// TwinCAT 3 PLC project DCSv1
// ProgramVersion: 3.1.4023.0
// libraries:
//   Tc2_MC2, * (Beckhoff Automation GmbH)
//   Tc2_MC2_Drive, * (Beckhoff Automation GmbH)
//   Tc2_SerialCom, * (Beckhoff Automation GmbH)
//   Tc2_Standard, * (Beckhoff Automation GmbH)
//   Tc2_System, * (Beckhoff Automation GmbH)
//   Tc3_Module, * (Beckhoff Automation GmbH)
// project tree:
//   / ComTask.TcTTO (not stored), PlcTask.TcTTO (not stored)
//   GVLs/GVLs/ GVL.TcGVL, GVL_IO.TcGVL, GVL_ResearchData.TcGVL, GVL_VAR.TcGVL, ReadMe.TcGVL
//   POUs/FB/ FB_Analog.TcPOU (not stored), F_ScalAnalogOut.TcPOU
//   POUs/ MAIN.TcPOU, P_AP1_Check.TcPOU, P_ComEL6001.TcPOU (not stored), P_CP1_Calibration.TcPOU, P_CP1_Enable.TcPOU (not stored), P_MI1_OnOff.TcPOU (not stored), P_AP1_OnOff.TcPOU (not stored), P_ModeSelector.TcPOU, P_Outputs_Manual.TcPOU, P_Set_Research_Data.TcPOU, P_Read_Research_Data.TcPOU, P_SP1_Check.TcPOU, P_SP1_OnOff.TcPOU
//   POUs/POUs/ FB_Drive.TcPOU (not stored), FB_Mixer1_2.TcPOU
// real-time tasks:
//   TASK PlcTask: cycle T#10ms, priority 20, ADS port 350
//   TASK ComTask: cycle T#10ms, priority 21, ADS port 351
// motion (NC):
//   TASK NC-Task 1 SAF: cycle T#2ms, priority 4, ADS port 501
//   TASK NC-Task 1 SVB: cycle T#10ms, priority 8, ADS port 511
//   AXIS Mixer 1 (id 2)
//     General: UnitName=°, UnitFlags=#x00000004
//     Dynamic: Acceleration=7443.34, Deceleration=7443.34, Jerk=22330
//     Velo: RefSearch=49.6222741699219, RefSync=49.6222741699219, SlowManual=248.111370849609, FastManual=1488.66822509766, Fast=4962.22741699219, Maximum=4962.23
//     OtherSettings: AllowMotionCmdToSlave=true
//     encoder EncType=8
//       EncPara: ScaleFactorNumerator=45, ScaleFactorDenominator=1048576, Offset=-131121.7408, Inverse=true, MaxCount=#x007fffff, ReferenceSystem=2
//     drive DrvType=9
//       DrvPara: Inverse=true, MaxCount=#xffffffff, DriveControlDWord=#x00030100
//         Analog: VeloReferenz=5458.45015869141, VeloScale=1.02400649589962, ScaleFactorActTorque=0.1
//         TimeComp: TaskDelayCycles=1
//     controller CtrType=1
//       CtrPara: PriorControlFactor=1
//         Observer: BandWidth=20
//   AXIS Mixer 2 (id 3)
//     General: UnitName=°, UnitFlags=#x00000004
//     Dynamic: Acceleration=7443.34112548828, Deceleration=7443.34112548828, Jerk=22330.0233764648
//     Velo: RefSearch=49.6222741699219, RefSync=49.6222741699219, SlowManual=248.111370849609, FastManual=1488.66822509766, Fast=4962.22741699219, Maximum=4962.22741699219
//     OtherSettings: AllowMotionCmdToSlave=true
//     encoder EncType=8
//       EncPara: ScaleFactorNumerator=45, ScaleFactorDenominator=1048576, MaxCount=#x007fffff, ReferenceSystem=2
//     drive DrvType=9
//       DrvPara: MaxCount=#xffffffff, DriveControlDWord=#x00030100
//         Analog: VeloReferenz=5458.45015869141, VeloScale=1.02400649589962, ScaleFactorActTorque=0.1
//         TimeComp: TaskDelayCycles=1
//     controller CtrType=1
//       CtrPara: PriorControlFactor=1
//         Observer: BandWidth=20
// I/O:
//   DEVICE Device 1 (EtherCAT), AmsNetId 172.17.147.1.3.1
//     Term 1 (EK1200) [EK1200-5000 EtherCAT Power supply (2A E-Bus)]
//       Term 2 (EL1008) 30K3 [EL1008 8Ch. Dig. Input 24V, 3ms]
//       Term 3 (EL1008) 30K3.1 [EL1008 8Ch. Dig. Input 24V, 3ms]
//       Term 10 (EL1008) new [EL1008 8Ch. Dig. Input 24V, 3ms]
//       Term 4 (EL2008) 30K4 [EL2008 8Ch. Dig. Output 24V, 0.5A]
//       Term 5 (EL2008) 30K5 [EL2008 8Ch. Dig. Output 24V, 0.5A]
//       Term 12 (EL2008) new [EL2008 8Ch. Dig. Output 24V, 0.5A]
//       Term 13 (EL3022) new [EL3022 2Ch. Ana. Input 4-20mA DIFF]
//       Term 14 (EL3202) new [EL3202 2Ch. Ana. Input PT100 (RTD)]
//       Term 6 (EL3255) 30K5.1 [EL3255 5Ch. potentiometer measurement with sensor supply]
//       Term 7 (EL4134) 30K6 [EL4134 4Ch. Ana. Output -10/+10V, 16bit]
//       Term 8 (EL6001) [EL6001 Interface (RS232)]
//       Term 15 (EL6631) new [EL6631 PROFINET IO Controller]
//       Term 9 (EL9011) [EL9011 End Terminal]
//   DEVICE Device 4 (EtherCAT), AmsNetId 172.17.147.1.5.1
//     Drive 11 (AX5206-0000-0213) [AX5206-0000-0213 EtherCAT Drive (SoE, 2 Ch.)]
// variable links:
//   NC-Task 1 SAF/Axes/Mixer 1 <-> Device 4 (EtherCAT)/Drive 11 (AX5206-0000-0213)
//     Drive/Inputs/In/nDataIn1 <-> AT 1/Following distance
//     Drive/Inputs/In/nDcOutputTime <-> InfoData/DcOutputShift
//     Drive/Inputs/In/nState1 <-> AT 1/Drive status word @bit 8
//     Drive/Inputs/In/nState2 <-> AT 1/Drive status word
//     Drive/Inputs/In/nState4 @bit 1 <-> WcState/InputToggle
//     Drive/Inputs/In/nState4 <-> WcState/WcState
//     Drive/Outputs/Out/nCtrl1 <-> MDT 1/Master control word @bit 8
//     Drive/Outputs/Out/nDataOut1 <-> MDT 1/Position command value
//     Enc/Inputs/In/nDataIn1 <-> AT 1/Position feedback 1 value
//     Enc/Inputs/In/nDcInputTime <-> InfoData/DcInputShift
//     Enc/Inputs/In/nState4 @bit 1 <-> WcState/InputToggle
//     Enc/Inputs/In/nState4 <-> WcState/WcState
//   NC-Task 1 SAF/Axes/Mixer 2 <-> Device 4 (EtherCAT)/Drive 11 (AX5206-0000-0213)
//     Drive/Inputs/In/nDataIn1 <-> AT 2/Following distance
//     Drive/Inputs/In/nDcOutputTime <-> InfoData/DcOutputShift
//     Drive/Inputs/In/nState1 <-> AT 2/Drive status word @bit 8
//     Drive/Inputs/In/nState2 <-> AT 2/Drive status word
//     Drive/Inputs/In/nState4 @bit 1 <-> WcState/InputToggle
//     Drive/Inputs/In/nState4 <-> WcState/WcState
//     Drive/Outputs/Out/nCtrl1 <-> MDT 2/Master control word @bit 8
//     Drive/Outputs/Out/nDataOut1 <-> MDT 2/Position command value
//     Enc/Inputs/In/nDataIn1 <-> AT 2/Position feedback 1 value
//     Enc/Inputs/In/nDcInputTime <-> InfoData/DcInputShift
//     Enc/Inputs/In/nState4 @bit 1 <-> WcState/InputToggle
//     Enc/Inputs/In/nState4 <-> WcState/WcState
//   DCSv1/DCSv1 Instance <-> Device 1 (EtherCAT)/Term 1 (EK1200)/Term 10 (EL1008) new
//     PlcTask Inputs/GVL_IO.ib_SP1_No_Error <-> Channel 2/Input
//     PlcTask Inputs/GVL_IO.ib_SP1_Ready <-> Channel 1/Input
//   DCSv1/DCSv1 Instance <-> Device 1 (EtherCAT)/Term 1 (EK1200)/Term 2 (EL1008) 30K3
//     ComTask Inputs/GVL_IO.ib_CP1_Ready <-> Channel 3/Input
//     PlcTask Inputs/GVL_IO.ib_AP1_No_Error <-> Channel 6/Input
//     PlcTask Inputs/GVL_IO.ib_AP1_Ready <-> Channel 5/Input
//     PlcTask Inputs/GVL_IO.ib_CC1_Button_Mode_Laptop <-> Channel 8/Input
//     PlcTask Inputs/GVL_IO.ib_CC1_Button_Reset <-> Channel 7/Input
//     PlcTask Inputs/GVL_IO.ib_CC1_Safety_Ready <-> Channel 1/Input
//     PlcTask Inputs/GVL_IO.ib_CP1_Drive_Error <-> Channel 4/Input
//     PlcTask Inputs/GVL_IO.ib_CP1_Safety_Grid_Mounted <-> Channel 2/Input
//   DCSv1/DCSv1 Instance <-> Device 1 (EtherCAT)/Term 1 (EK1200)/Term 3 (EL1008) 30K3.1
//     PlcTask Inputs/GVL_IO.ib_AP1_Button_Not_Off <-> Channel 7/Input
//     PlcTask Inputs/GVL_IO.ib_AP1_Button_On <-> Channel 6/Input
//     PlcTask Inputs/GVL_IO.ib_CC1_Button_Mode_Manual <-> Channel 1/Input
//     PlcTask Inputs/GVL_IO.ib_MI1_Button_Not_Off <-> Channel 3/Input
//     PlcTask Inputs/GVL_IO.ib_MI1_Button_On <-> Channel 2/Input
//     PlcTask Inputs/GVL_IO.ib_SP1_Button_Not_Off <-> Channel 5/Input
//     PlcTask Inputs/GVL_IO.ib_SP1_Button_On <-> Channel 4/Input
//   DCSv1/DCSv1 Instance <-> Device 1 (EtherCAT)/Term 1 (EK1200)/Term 4 (EL2008) 30K4
//     PlcTask Outputs/GVL_IO.ob_AP1_Pressure_Ok <-> Channel 7/Output
//     PlcTask Outputs/GVL_IO.ob_AP1_Pulse <-> Channel 8/Output
//     PlcTask Outputs/GVL_IO.ob_AP1_Start <-> Channel 6/Output
//     PlcTask Outputs/GVL_IO.ob_CC1_Safety_Reset <-> Channel 1/Output
//     PlcTask Outputs/GVL_IO.ob_CP1_Backward <-> Channel 5/Output
//     PlcTask Outputs/GVL_IO.ob_CP1_Forward <-> Channel 4/Output
//     PlcTask Outputs/GVL_IO.ob_CP1_Start <-> Channel 3/Output
//     PlcTask Outputs/GVL_IO.ob_CP1_Stop <-> Channel 2/Output
//   DCSv1/DCSv1 Instance <-> Device 1 (EtherCAT)/Term 1 (EK1200)/Term 5 (EL2008) 30K5
//     PlcTask Outputs/GVL_IO.ob_AP1_Not_Empty <-> Channel 1/Output
//     PlcTask Outputs/GVL_IO.ob_AP1_Power_On <-> Channel 2/Output
//     PlcTask Outputs/GVL_IO.ob_SP1_Not_Empty <-> Channel 6/Output
//     PlcTask Outputs/GVL_IO.ob_SP1_Power_On <-> Channel 7/Output
//     PlcTask Outputs/GVL_IO.ob_SP1_Pressure_Ok <-> Channel 4/Output
//     PlcTask Outputs/GVL_IO.ob_SP1_Pulse <-> Channel 5/Output
//     PlcTask Outputs/GVL_IO.ob_SP1_Start <-> Channel 3/Output
//   DCSv1/DCSv1 Instance <-> Device 1 (EtherCAT)/Term 1 (EK1200)/Term 6 (EL3255) 30K5.1
//     ComTask Inputs/GVL_IO.in_AP1_Poti_Speed <-> AI Standard Channel 3/Value
//     ComTask Inputs/GVL_IO.in_PP1_Poti_Speed <-> AI Standard Channel 2/Value
//     PlcTask Inputs/GVL.nInputSpare1 <-> AI Standard Channel 4/Value
//     PlcTask Inputs/GVL.nInputSpare2 <-> AI Standard Channel 5/Value
//     PlcTask Inputs/GVL_IO.in_MI1_Poti_Speed <-> AI Standard Channel 1/Value
//   DCSv1/DCSv1 Instance <-> Device 1 (EtherCAT)/Term 1 (EK1200)/Term 7 (EL4134) 30K6
//     PlcTask Outputs/GVL_IO.on_AP1_Speed <-> AO Output Channel 2/Analog output
//     PlcTask Outputs/GVL_IO.on_CP1_Speed <-> AO Output Channel 1/Analog output
//     PlcTask Outputs/GVL_IO.on_SP1_Speed <-> AO Output Channel 3/Analog output
//   DCSv1/DCSv1 Instance <-> Device 1 (EtherCAT)/Term 1 (EK1200)/Term 8 (EL6001)
//     ComTask Inputs/GVL.stIn_EL6001/D <-> COM Inputs/Data In 0
//     ComTask Inputs/GVL.stIn_EL6001/D @bit {8..168 step 8} <-> COM Inputs/Data In {1..21}  (21 links)
//     ComTask Inputs/GVL.stIn_EL6001/Status <-> COM Inputs/Status
//     ComTask Outputs/GVL.stOut_EL6001/Ctrl <-> COM Outputs/Ctrl
//     ComTask Outputs/GVL.stOut_EL6001/D <-> COM Outputs/Data Out 0
//     ComTask Outputs/GVL.stOut_EL6001/D @bit {8..168 step 8} <-> COM Outputs/Data Out {1..21}  (21 links)
//   DCSv1/DCSv1 Instance <-> Device 4 (EtherCAT)/Drive 11 (AX5206-0000-0213)
//     PlcTask Inputs/GVL.in_MID1_ActAbsCurrent <-> AT 1/Actual absolute current
//     PlcTask Inputs/GVL.in_MID2_ActAbsCurrent <-> AT 2/Actual absolute current
//     PlcTask Inputs/GVL.in_MID1_ActMotorTemperature <-> AT 1/Motor temperature
//     PlcTask Inputs/GVL.in_MID2_ActMotorTemperature <-> AT 2/Motor temperature
//   DCSv1/DCSv1 Instance <-> NC-Task 1 SAF/Axes/Mixer 1
//     PlcTask Inputs/GVL.Axis_Mixer1.NcToPlc <-> Outputs/ToPlc
//     PlcTask Outputs/GVL.Axis_Mixer1.PlcToNc <-> Inputs/FromPlc
//   DCSv1/DCSv1 Instance <-> NC-Task 1 SAF/Axes/Mixer 2
//     PlcTask Inputs/GVL.Axis_Mixer2.NcToPlc <-> Outputs/ToPlc
//     PlcTask Outputs/GVL.Axis_Mixer2.PlcToNc <-> Inputs/FromPlc

// ---- GVLs/GVLs/GVL.TcGVL
{attribute 'qualified_only'}
VAR_GLOBAL
	
	
	//
	// Data Communication RS-232
	TxBufferEL								: ComBuffer;
	RxBufferEL								: ComBuffer;
	
			
	//
	// Data Communication Axis Mixers

	//
	// Mixer drive A // 16.09.2021 PF
	Axis_Mixer1 							: AXIS_REF;
	f_MID1_ActCurrent: REAL;
	f_MID1_ActTorque: REAL;
	in_MID1_ActAbsCurrent AT %I*: INT;
	in_MID1_ActMotorTemperature AT %I* :INT; // 220817 WT 
	
	//
	// Mixer drive B // 16.09.2021 PF
	Axis_Mixer2 							: AXIS_REF;
	f_MID2_ActCurrent: REAL;
	f_MID2_ActTorque: REAL;
	in_MID2_ActAbsCurrent AT %I*: INT;
	in_MID2_ActMotorTemperature AT %I* :INT; // 220817 WT
	
	//
	// Control Input Speed
	fControlMixerPumpSpeed					: REAL; 
	fControlPeristalticPumpSpeed			: REAL; 
	fControlDosingPumpSpeed					: REAL; 
	fInputSpare1							: REAL; 
	fInputSpare2							: REAL; 
	
	//
	// Output Speed
	fConcretePumpSpeed						: REAL;
	fDosingPumpSpeed						: REAL;
	fOutputSpare1							: REAL;
	fOutputSpare2							: REAL;
	
	
	//
	//Hardware Input
	bSafetyIO						AT %I*	: BOOL;
	// bConcretePumpSafetyGridMounted	AT %I*	: BOOL;
	// bConcretePumpReady				AT %I*	: BOOL;
	// bConcretePumpFcError				AT %I*	: BOOL;
	bDosingPumpReady				AT %I*	: BOOL;
	bDosingPumpNoError				AT %I*	: BOOL;
	bControlResetSafety				AT %I*	: BOOL;
	bControlLaptop					AT %I*	: BOOL;
	bControlManual					AT %I*	: BOOL;	
	nControlMixerPumpOn				AT %I*	: BOOL; 
	nControlMixerPumpOff			AT %I*	: BOOL; 
	nControlConcretPumpOn			AT %I*	: BOOL; 
	nControlConcretPumpOff			AT %I*	: BOOL; 
	nControlDosingPumpOn			AT %I*	: BOOL; 
	nControlDosingPumpOff			AT %I*	: BOOL; 
	bInputSpare1					AT %I*	: BOOL;
		
	nControlMixerPumpSpeed			AT %I*	: INT; 
	// nControlPeristalticPumpSpeed	AT %I*	: INT; 
	nControlDosingPumpSpeed			AT %I*	: INT; 
	nInputSpare1					AT %I*	: INT; 
	nInputSpare2					AT %I*	: INT; 

	
	//
	//Hardware Output
	bResetSafety					AT %Q*	: BOOL;
	// bConcretePumpOn					AT %Q*	: BOOL;
	// bConcretePumpOff					AT %Q*	: BOOL;
	// bConcretePumpForwardOn			AT %Q*	: BOOL;
	// bConcretePumpBackwardOn			AT %Q*	: BOOL;
	bDosingPumpDosingHighLow		AT %Q*	: BOOL;
	bDosingPumpNoFastStop			AT %Q*	: BOOL;
	bDosingPumpDosingAmount			AT %Q*	: BOOL;
	bOutputSpare1					AT %Q*	: BOOL;
	bOutputSpare2					AT %Q*	: BOOL;
	bOutputSpare3					AT %Q*	: BOOL;
	bOutputSpare4					AT %Q*	: BOOL;
	bOutputSpare5					AT %Q*	: BOOL;
	bOutputSpare6					AT %Q*	: BOOL;
	bOutputSpare7					AT %Q*	: BOOL;
	bOutputSpare8					AT %Q*	: BOOL;
	
	// nConcretePumpSpeed				AT %Q*	: INT;
	nDosingPumpSpeed				AT %Q*	: INT;
	nOutputSpare1					AT %Q*	: INT;
	nOutputSpare2					AT %Q*	: INT;
	
	
	//
	//Hardware RS-232
	stIn_EL6001 					AT %I*	: EL6inData22B;	
	stOut_EL6001 					AT %Q*	: EL6outData22B;
	
END_VAR

// ---- GVLs/GVLs/GVL_IO.TcGVL
{attribute 'qualified_only'}
VAR_GLOBAL
//***********************************************************************************
//
// ETH Zürich / Robotic Fabrication Lab
// HIB C 13 / Stefano-Franscini-Platz 1
// CH-8093 Zürich
// 
// ***********************************************************************************
// 
// PROJECT     :  A061 Inline Mixer
// 
// FUNCTION    :  Global Varable In and Outputs
// 
// AUTHOR      :  Fabio Scotto / Philippe Fleischmann
// 
// EMAIL       :  scotto@arch.ethz.ch / fleischmann@arch.ehtz.ch
// 
// Copyright   :  ETH Zürich (CH) 2020
//
// ***********************************************************************************

//
// Inputs

//
// Concrete Controller 1
ib_CC1_Safety_Ready AT %I*: BOOL;
ib_CC1_Button_Mode_Manual AT %I*: BOOL;
ib_CC1_Button_Mode_Laptop AT %I*: BOOL;
//ib_CC1_Button_Mode_Robot AT %I*:BOOL;
//
ib_CC1_Button_Reset AT %I*: BOOL;

//
// Concrete Pump 1
ib_CP1_Drive_Error AT %I*: BOOL;
ib_CP1_Ready AT %I*: BOOL;
ib_CP1_Safety_Grid_Mounted AT %I*: BOOL;
in_CP1_Tube_Pressure_Sensor AT %I*: INT;
in_CP1_Tube_Temperature_Sensor AT %I*: INT;

//
// Peristaltic Pump 1 ( SHOULD BE REMOVE, it is old pump 
in_PP1_Poti_Speed AT %I*	: INT; 

//
// Accelerator Pump 1
ib_AP1_Button_On AT %I*: BOOL;
ib_AP1_Button_Not_Off AT %I*: BOOL;
ib_AP1_Ready AT %I*: BOOL;
ib_AP1_No_Error AT %I*: BOOL;
in_AP1_Poti_Speed AT %I*	: INT; 

// 
// Superplasticizer Pump 1 (WT 220915)
ib_SP1_Button_On AT %I*: BOOL;
ib_SP1_Button_Not_Off AT %I*: BOOL;
ib_SP1_Ready AT %I*: BOOL;
ib_SP1_No_Error AT %I*: BOOL;
ib_SP1_Poti_Speed AT %I*: INT; 

//
// Mixer 1
ib_MI1_Button_On AT %I*: BOOL;
ib_MI1_Button_Not_Off AT %I*: BOOL;
in_MI1_Poti_Speed AT %I*	: INT; 

//
// Outputs

//
// Concrete Controller 1
ob_CC1_Safety_Reset AT %Q*: BOOL;

//
// Concrete Pump 1
ob_CP1_Start AT %Q*: BOOL;
ob_CP1_Stop AT %Q*: BOOL;
ob_CP1_Forward AT %Q*: BOOL;
ob_CP1_Backward AT %Q*: BOOL;

on_CP1_Speed AT %Q*: INT;

//
// Accelerator Pump 1
ob_AP1_Power_On AT %Q*: BOOL;
ob_AP1_Start AT %Q*: BOOL;
ob_AP1_Pressure_Ok AT %Q*: BOOL;
ob_AP1_Not_Empty AT %Q*: BOOL;
ob_AP1_Pulse AT %Q*: BOOL;

on_AP1_Speed AT %Q*: INT;

// 
// Superplasticizer Pump 1 (WT 220915)
ob_SP1_Power_On AT %Q*: BOOL;
ob_SP1_Start AT %Q*: BOOL;
ob_SP1_Pressure_Ok AT %Q*: BOOL;
ob_SP1_Not_Empty AT %Q*: BOOL;
ob_SP1_Pulse AT %Q*: BOOL;

on_SP1_Speed AT %Q*: INT;


END_VAR

// ---- GVLs/GVLs/GVL_ResearchData.TcGVL
{attribute 'qualified_only'}
VAR_GLOBAL
//***********************************************************************************
//
// ETH Zürich / Robotic Fabrication Lab
// HIB C 13 / Stefano-Franscini-Platz 1
// CH-8093 Zürich
// 
// ***********************************************************************************
// 
// PROJECT     :  A061 Inline Mixer
// 
// FUNCTION    :  Global Varable to collect all research data
// 
// AUTHOR      :  Seyma Gürel / Philippe Fleischmann / Weiting Chen
// 
// EMAIL       :  scotto@arch.ethz.ch / fleischmann@arch.ehtz.ch
// 
// Copyright   :  ETH Zürich (CH) 2021
//
// ***********************************************************************************


// ***********************************************************************************
// Process inputs
// ***********************************************************************************

//
// Mode
b_RED_Mode_Manual: BOOL; //0916 WT
b_RED_Mode_Laptop: BOOL; //0916 WT

//
// Maximal speed for mixer [°/s]  (WT 220916
f_RED_Control_Speed : LREAL;					// [°/s]
b_RED_Laptop_speed_Conctrol: BOOL;
f_RED_Control_Speed_by_Laptop:LREAL;

//
Superplasticizer_Pump: STRING := 'Superplasticizer_Pump'; 
// 
// Superplasticizer Pump (WT 220916 
b_RED_Superplasticizer_Pump_Check_On: BOOL;
n_RED_Superplasticizer_Pump_Check_Flowrate: REAL;
n_RED_Superplasticizer_Pump_Check_Duration: TIME;

b_RED_Superplasticizer_Pump_Flush_On: BOOL;
n_RED_Superplasticizer_Pump_Flush_Speed: REAL;

f_RED_Superplasticizer_Pump_Mass: REAL;             // [g/min]
f_RED_Superplasticizer_Pump_Density: REAL;          // [g/ml]
n_RED_Superplasticizer_Pump_Flowrate: REAL;         // [ml/min]

//
ACCELERATION_PUMP: STRING := 'Acceleration_Pump';
//
// Accelerator Pump
b_RED_Acceleration_Pump_Check_On: BOOL;
n_RED_Acceleration_Pump_Check_Flowrate: REAL;
n_RED_Acceleration_Pump_Check_Duration: TIME;

b_RED_Acceleration_Pump_Flush_On: BOOL;
n_RED_Acceleration_Pump_Flush_Speed: REAL;

f_RED_Acceleration_Pump_Mass: REAL;             // [g/min]
f_RED_Acceleration_Pump_Density: REAL;          // [g/ml]
n_RED_Acceleration_Pump_Flowrate: REAL;         // [ml/min]

//
CONCRETE_PUMP: STRING := 'CONCRETE_PUMP';
// Concrete Pump
//
b_RED_Concrete_Pump_Forward_On: BOOL;
b_RED_Concrete_Pump_Backward_On: BOOL;
n_RED_Concrete_Pump_Speed: INT;					// [ 0..75rpm ]
// WT 220916
b_RED_Concrete_Pump_Calibration_On: BOOL;
n_RED_Concrete_Pump_Calibration_Speed: INT;		// [rpm]
n_RED_Concrete_Pump_Calibration_Time: TIME;


// ***********************************************************************************
// Process outpus
// ***********************************************************************************

//
MIXER: STRING := 'MIXER';
// Status mixer
//
b_RED_Status_On : BOOL;
f_RED_Status_Speed_Overide : LREAL;
f_RED_Status_Speed_Motor_1 : LREAL;
f_RED_Status_Speed_Motor_2 : LREAL;
f_RED_Status_Torque_Motor_1 : REAL;				// [Nm]
f_RED_Status_Torque_Motor_2 : REAL;				// [Nm]

f_RED_Status_Temperature_Motor_1 : REAL; // [°C] 
f_RED_Status_Temperature_Motor_2 : REAL; // [°C] 

//
// Superplasticizer Pump (WT 220916
n_RED_Status_Superplasticizer_Pump_Flowrate: INT;          // [ml/min]
f_RED_Status_Superplasticizer_Pump_Max_Flowrate_ml_per_min: REAL;           // [ml/min]

//
// Accelerator Pump
n_RED_Status_Acceleration_Pump_Flowrate: INT;          // [ml/min]
f_RED_Status_Acceleration_Pump_Max_Flowrate_ml_per_min: REAL;           // [ml/min]

	n_RED_Acceleration_Pump_Calibration_Speed: INT;
	b_RED_Acceleration_Pump_Preparation_On: INT;
END_VAR

// ---- GVLs/GVLs/GVL_VAR.TcGVL
{attribute 'qualified_only'}
VAR_GLOBAL
//***********************************************************************************
//
// ETH Zürich / Robotic Fabrication Lab
// HIB C 13 / Stefano-Franscini-Platz 1
// CH-8093 Zürich
// 
// ***********************************************************************************
// 
// PROJECT     :  A061 Inline Mixer
// 
// FUNCTION    :  Global Varable In and Outputs
// 
// AUTHOR      :  Fabio Scotto / Philippe Fleischmann / Weiting Chen
// 
// EMAIL       :  scotto@arch.ethz.ch / fleischmann@arch.ehtz.ch
// 
// Copyright   :  ETH Zürich (CH) 2020
//
// ***********************************************************************************

//
// Concrete Controller 1
b_Mode_Manual : BOOL;
b_Mode_Laptop : BOOL;

//
// Concrete Pump 1

//
// Superplasticizer Pump 1
b_SP1_Run : BOOL;
f_SP1_Override :LREAL;

//
// Accelerator Pump 1
b_AP1_Run : BOOL;
f_AP1_Override : LREAL; 

//
// Mixer 1
b_MI1_ReadToDrive : BOOL;
b_MI1_Run : BOOL;
f_MI1_Override : LREAL; 
f_MI1_MaxSpeed : LREAL;
f_MI1_ActSpeedM1 : LREAL;
f_MI1_ActSpeedM2 : LREAL;

END_VAR

// ---- GVLs/GVLs/ReadMe.TcGVL
{attribute 'qualified_only'}
VAR_GLOBAL
//***********************************************************************************
//
// ETH Zürich / Robotic Fabrication Lab
// HIB C 13 / Stefano-Franscini-Platz 1
// CH-8093 Zürich
// 
// ***********************************************************************************
// 
// PROJECT     :  A061 Inline Mixer
// 
// FUNCTION    :  Read Me
// 
// AUTHOR      :  Fabio Scotto / Philippe Fleischmann
// 
// EMAIL       :  scotto@arch.ethz.ch / fleischmann@arch.ehtz.ch
// 
// Copyright   :  ETH Zürich (CH) 2020
//
// ***********************************************************************************

//
//Prefix
//ib = Input Bool   / ob = Output Bool
//if = Input float  / of = Output float (REAL, LREAL)
//in = Input numeric/ on = Outplut numerical (INT, Sint, USINT, UNIT, DINT, UDINT, BYTE, WORD, DWORD, LWORD, XINT, UXINT, XWORD) 

//
//Short Cuts
//CC1 = Concrete Controller 
//AP1 = Accelerator Pump
//CP1 = Concrete Pump
//PP1 = Peristaltic Pump
//MI1 = Mixer
//T1  = Tool 1
//CA1 = Camera 1
//RED = Research Data

END_VAR

// ---- POUs/FB/F_ScalAnalogOut.TcPOU
FUNCTION F_ScalAnalogOut : INT
VAR_INPUT
	n_Input:INT;
	n_InMin:INT;
	n_InMax:INT;
	n_OutMin:INT;
	n_OutMax:INT;

END_VAR
VAR
	f_Input:REAL;
	f_InMin:REAL;
	f_InMax:REAL;
	f_OutMin:REAL;
	f_OutMax:REAL;
	f_DeltaIn:REAL;
	f_DeltaOut:REAL;
END_VAR

//
// Convert integer to real 
f_Input:=INT_TO_REAL(n_Input);
f_InMin:=INT_TO_REAL(n_InMin);
f_InMax:=INT_TO_REAL(n_InMax);
f_OutMin:=INT_TO_REAL(n_OutMin);
f_OutMax:=INT_TO_REAL(n_OutMax);
//
// Check plausibility 
IF f_InMax = f_InMin THEN	
	//
	// Not plausible output fix value
	F_ScalAnalogOut := 0;
ELSE	
	//
	// Plausible calculate output 
	f_DeltaIn:=f_InMax-f_InMin;
	f_DeltaOut:=f_OutMax-f_OutMin;
	F_ScalAnalogOut :=REAL_TO_INT((f_DeltaOut/f_DeltaIn)*(f_Input-f_InMin));	
END_IF

END_FUNCTION

// ---- POUs/MAIN.TcPOU
PROGRAM MAIN
VAR	

	fb_MC_SetPosition		:FB_SoEAX5000SetPositionOffset;
	pos:LREAL;
	Mixer1_2		: FB_Mixer1_2;
	Analog			: FB_Analog;

	SafetyReset 	: bool;
	b_Enable		: BOOL;
	b_Reset			: BOOL;


	
	Test : MC_ReadStatus;
END_VAR

//***********************************************************************************
//
// ETH Zürich / Robotic Fabrication Lab
// HIB C 13 / Stefano-Franscini-Platz 1
// CH-8093 Zürich
// 
// ***********************************************************************************
// 
// PROJECT     :  A061 Inline Mixer
// 
// FUNCTION    :  MAIN Programm
// 
// AUTHOR      :  Mathias Suter /Weiting Chen
// 
// EMAIL       :  mathias.suter@solinaut.ch
// 
// Copyright   :  ETH Zürich (CH) 2021
//
// ***********************************************************************************


//
// Mode selector ( ONLY FOR READ OUTPUT NOW
P_ModeSelector();

//
// Set research data 
P_Set_Research_Data();

// ******************************************************************
// 220916 WT

//*************************
// Superplasticizer Pump
//*************************

//
// Superplasticizer Pump 1 Calibraration (220916 WT
P_SP1_Check();

//
// Superplasticizer Pump 1 On/Off
IF GVL_ResearchData.b_RED_Superplasticizer_Pump_Check_On=FALSE THEN
	//
	// Superplasticizer Pump 1 On/Off
	P_SP1_OnOff();
END_IF

//*************************
// Acceleration Pump
//*************************

//
// Acceleration Pump 1 Calibraration
P_AP1_Check();

//
// Check for Acceleration Pump 1 state
IF GVL_ResearchData.b_RED_Acceleration_Pump_Check_On=FALSE THEN
	//
	// Acceleration Pump 1 On/Off 
	P_AP1_OnOff();
END_IF

//*************************
// Concrete Pump
//*************************


// ******************************************************************
//
// Mixer On/Off 
P_MI1_OnOff();

//
// Temporary scaling of the poti and laptop ontrol for the mixer override  (WT 220916
IF GVL_ResearchData.b_RED_Laptop_speed_Conctrol THEN
	IF GVL_ResearchData.f_RED_Control_Speed_by_Laptop > 100
		THEN
		GVL_ResearchData.f_RED_Control_Speed_by_Laptop:=100;
	END_IF
	GVL_VAR.f_MI1_Override:=GVL_ResearchData.f_RED_Control_Speed_by_Laptop;
ELSE
	GVL_VAR.f_MI1_Override:=100.0 / 32767 * GVL_IO.in_MI1_Poti_Speed;
END_IF


//
// Mixer 1 + 2
Mixer1_2(
	Mixer1			:= GVL.Axis_Mixer1,
 	Mixer2			:= GVL.Axis_Mixer2,
	f_Velocity		:= GVL_VAR.f_MI1_MaxSpeed,
	b_JogForward	:= FALSE,
	b_JogBackwards	:= GVL_VAR.b_MI1_Run,
 	b_Enable		:= GVL_IO.ib_CC1_Button_Mode_Manual AND GVL_IO.ib_CC1_Safety_Ready,	
 	b_Reset			:= GVL_IO.ib_CC1_Button_Reset,
	f_Override		:= GVL_VAR.f_MI1_Override);	
	(*
	fb_MC_SetPosition(
	Axis			:= GVL.Axis_Mixer2,
	memory			:= 1,
	Feedback		:= 0);*)
	
pos:=GVL.Axis_Mixer2.NcToPlc.ModuloActPos;


//
GVL.f_MID1_ActCurrent:=GVL.in_MID1_ActAbsCurrent * 5.9 / 1000;
GVL.f_MID1_ActTorque:=GVL.f_MID1_ActCurrent * 0.8 * 8; // Torque constante / Gear transaltion

GVL.f_MID2_ActCurrent:=gvl.in_MID2_ActAbsCurrent * 5.9 / 1000;
GVL.f_MID2_ActTorque:=GVL.f_MID2_ActCurrent * 0.8 * 8; // Torque constante / Gear transaltion

//
// Write global variable for mixer ready to drive
GVL_VAR.b_MI1_ReadToDrive:=Mixer1_2.b_ReadyToDrive;
	
// 
// Reset 
GVL_IO.ob_CC1_Safety_Reset:=GVL_IO.ib_CC1_Button_Reset;
 	
// GVL.bResetSafety	:= safetyReset;


//
// Concrete pump
P_CP1_Enable();
	
// Analog();

//
// Outputs
P_Outputs_Manual();

//
// Read researchs data 
P_Read_Research_Data();

END_PROGRAM

// ---- POUs/POUs/FB_Mixer1_2.TcPOU
FUNCTION_BLOCK FB_Mixer1_2
VAR_INPUT
	// General
	b_Enable				: BOOL;		
	b_Reset					: BOOL;
	
	// Parameter SetPosition
	b_ModeSetPosition		: BOOL;				// Active Mode SetPosition
	b_SetPositionMixer1		: BOOL;				// SetPositon mixer 1 with f_SetPosition1
	b_SetPositionMixer2		: BOOL;				// SetPositon mixer 2 with f_SetPosition1
	f_SetPositionMixer1		: LREAL;			
	f_SetPositionMixer2		: LREAL;			
	
	//Parameter positions
	f_OffsetPositionMixer1 	: LREAL;			// 0..360°
	f_OffsetPositionMixer2 	: LREAL;			// 0..360°	
	f_CollisionPosMin		: LREAL := 35; 		// 0°..f_CollisionPosMax
	f_CollisionPosMax		: LREAL	:= 145;		// f_CollisionPosMin..180°
	f_OffsetMixer1Mixer2	: LREAL := 90; 		//0..360°
	
	//
	// Parameter drive
	f_Override				: LREAL;
	f_Velocity				: LREAL;
	b_JogForward			: BOOL;
	b_JogBackwards			: BOOL;
END_VAR
VAR_OUTPUT
	b_PowerActiveMixer1		: BOOL;
	b_PowerActiveMixer2		: BOOL;
	b_ReadyToDrive			: BOOL;
	b_ErrorGen				: BOOL;
	b_ErrorMixer1			: BOOL;
	b_ErrorMixer2			: BOOL;
	n_ErrorIDMixer1			: UDINT;
	n_ErrorIDMixer2			: UDINT;
	f_ActVelocityMixer1		: LREAL;
	f_ActVelocityMixer2		: LREAL;
	f_ActTorqueMixer1		: LREAL;
	f_ActTorqueMixer2		: LREAL;
	f_ActPositionMixer1		: LREAL;
	f_ActPositionMixer2		: LREAL;
END_VAR
VAR_IN_OUT
	Mixer1					: AXIS_REF;
	Mixer2					: AXIS_REF;
END_VAR
VAR		
	n_Step					: INT;				// Step chain
	b_ErrorInt				: BOOL;				// Error Intern

	b_Mixer1InCollision		: BOOL;				// Check if paddle mixer 1 in collision zone
	b_Mixer2InCollision		: BOOL;				// Check if paddle mixer 2 in collision zone
	f_PositionMixer1		: LREAL; 			// Position paddle mixer 1 in 0°..180°
	f_PositionMixer2		: LREAL; 			// Position paddle mixer 2 in 180°..360° (scaled 180°..0°)                                               
	f_ActPositionMixer1Calc	: LREAL;			// Actual position mixer 1 (with offset)
	f_ActPositionMixer2Calc	: LREAL;			// Actual position mixer 2 (with offset)

	// FBs	
	fb_Mixer1				: FB_Drive;	
	fb_Mixer2				: FB_Drive;	
	fb_MC_GearIn			: MC_GearIn;
	fb_MC_GearOut			: MC_GearOut;	
	fb_MC_ReadStatusMixer1	: MC_ReadStatus;
	fb_MC_ReadStatusMixer2	: MC_ReadStatus;
END_VAR

//***********************************************************************************
//
// ETH Zürich / Robotic Fabrication Lab
// HIB C 13 / Stefano-Franscini-Platz 1
// CH-8093 Zürich
// 
// ***********************************************************************************
// 
// PROJECT     :  ?? 
// 
// FUNCTION    :  FB_DriveGea
// 
// AUTHOR      :  Mathias Suter
// 
// EMAIL       :  mathias.suter@solinaut.ch
// 
// Copyright   :  ETH Zürich (CH) 2021
//
// ***********************************************************************************

//
// Limit f_OffsetPositionMixer1 and f_OffsetPositionMixer2 to 0°..360°
IF f_OffsetPositionMixer1 < 0 THEN
	f_OffsetPositionMixer1 := 0;
END_IF
IF f_OffsetPositionMixer1 > 360 THEN
	f_OffsetPositionMixer1 := 360;
END_IF

IF f_OffsetPositionMixer2 < 0 THEN
	f_OffsetPositionMixer2 := 0;
END_IF
IF f_OffsetPositionMixer2 > 360 THEN
	f_OffsetPositionMixer2 := 360;
END_IF

//
// Calculate and limit f_ActPosition1Calc and f_ActPosition1Calc to 0°..360°
f_ActPositionMixer1Calc := f_ActPositionMixer1 + f_OffsetPositionMixer1;
IF f_ActPositionMixer1Calc < 0 THEN
	f_ActPositionMixer1Calc := f_ActPositionMixer1Calc + 360;
ELSIF f_ActPositionMixer1Calc > 360 THEN
	f_ActPositionMixer1Calc := f_ActPositionMixer1Calc - 360;
END_IF

f_ActPositionMixer2Calc := f_ActPositionMixer2 + f_OffsetPositionMixer2;
IF f_ActPositionMixer2Calc < 0 THEN
	f_ActPositionMixer2Calc := f_ActPositionMixer1Calc + 360;
ELSIF f_ActPositionMixer2Calc > 360 THEN
	f_ActPositionMixer2Calc := f_ActPositionMixer1Calc - 360;
END_IF

//
// Calculate which position has the mixer 1 paddle in 0°-180° zone (f_ActPosition1Calc or f_ActPosition1Calc + 180°)
// for checking collision
IF f_ActPositionMixer1Calc < 180 THEN
	f_PositionMixer1 := f_ActPositionMixer1Calc;
ELSE	
	f_PositionMixer1 := f_ActPositionMixer1Calc - 180;
END_IF

//
// Calculate which position has the mixer 1 paddle in 180°-360° zone (f_ActPosition2Calc or f_ActPosition2Calc + 180°) 
// scale position 180° - 360° to 180° - 0°, for checking collision
(*IF f_ActPositionMixer2Calc < 180 THEN
	f_PositionMixer2 := 180 - f_ActPositionMixer2Calc;
ELSE	
	f_PositionMixer2 := 360 - f_ActPositionMixer2Calc;
END_IF*)

IF f_ActPositionMixer2Calc < 180 THEN
	f_PositionMixer2 := f_ActPositionMixer2Calc;
ELSE	
	f_PositionMixer2 := f_ActPositionMixer2Calc - 180;
END_IF

//
//Check if paddle in collision zone
b_Mixer1InCollision := f_PositionMixer1 > f_CollisionPosMin AND f_PositionMixer1 < f_CollisionPosMax;
b_Mixer2InCollision := f_PositionMixer2 > f_CollisionPosMin AND f_PositionMixer2 < f_CollisionPosMax;

//
// Limit offset mixer 1 to mixer 2 (for driving)
IF f_OffsetMixer1Mixer2 < 0 THEN
	f_OffsetMixer1Mixer2 := 0;
END_IF
IF f_OffsetMixer1Mixer2 > 360 THEN
	f_OffsetMixer1Mixer2 := 360;
END_IF

fb_MC_ReadStatusMixer1(Axis:=Mixer1,
					Enable:=TRUE);

fb_MC_ReadStatusMixer2(Axis:=Mixer2,
					Enable:=TRUE);


//
// Step chain for Gear In two Axis
CASE n_step OF
	
	0:
		//
		// Init
		n_Step := 10;
	
	10:
		//
		// Enable or set position
		IF b_Enable THEN
			n_Step := 20;
		END_IF;
		
		//
		// Error
		IF b_ErrorInt THEN
			n_Step := 200;
		END_IF
			
	20:
		//
		// GearOut
		IF fb_MC_GearOut.Done THEN
			n_Step := 30;
		END_IF
		
		//
		// Not Enable or Error	
		IF NOT b_Enable THEN
			n_Step := 10;
 		ELSIF b_ErrorInt THEN
			n_Step := 200;
		END_IF

	30:
		//
		//Set position posible (via b_SetPosition1 or b_SetPosition2 to value f_SetPosition1/f_SetPosition2)
				
		//
		// End set position 
		IF NOT b_ModeSetPosition THEN
			n_Step := 35;
		END_IF
			
		//
		// Not Enable or Error	
		IF NOT b_Enable THEN
			n_Step := 10;
 		ELSIF b_ErrorInt THEN
			n_Step := 200;
		END_IF
	35:
		//
		//Enable
		IF fb_Mixer1.b_PowerActive AND fb_Mixer2.b_PowerActive THEN
			n_Step := 40;	
		END_IF
		
		//
		// Not Enable or Error	
		IF NOT b_Enable THEN
			n_Step := 10;
 		ELSIF b_ErrorInt THEN
			n_Step := 200;
		END_IF
		
	40:
		//
		// Check mixer 1 or mixer 2 in collision zone
		IF b_Mixer1InCollision OR b_Mixer1InCollision THEN
			IF f_PositionMixer1 < f_PositionMixer2 THEN 
				//
				// Drive backwards out off collision zone
				n_Step := 50;
			ELSE
				//
				// Drive forward  out off collision zone
				n_Step := 60;
			END_IF;
		ELSE
			//
			// No driving
			n_Step := 70;
		END_IF
		
		//
		// Not Enable or Error	
		IF NOT b_Enable THEN
			n_Step := 10;
 		ELSIF b_ErrorInt THEN
			n_Step := 200;
		END_IF
		
	50:
		//
		// Drive till mixer 1 and mixer 2 not in collision zone (drive backwards)
		IF NOT b_Mixer1InCollision AND NOT b_Mixer2InCollision THEN
			n_Step := 70;
		END_IF
				
		//
		// Not Enable or Error	
		IF NOT b_Enable THEN
			n_Step := 10;
 		ELSIF b_ErrorInt THEN
			n_Step := 200;
		END_IF

	60:
		//
		// Drive till mixer 1 and mixer 2 not in collision zone (drive forward)
		IF NOT b_Mixer1InCollision AND NOT b_Mixer2InCollision THEN
			n_Step := 70;
		END_IF
		
		//
		// Not Enable or Error	
		IF NOT b_Enable THEN
			n_Step := 10;
 		ELSIF b_ErrorInt THEN
			n_Step := 200;
		END_IF
					
	70:
		//
		// Check mixer 1 and mixer 2 standstill
		IF Mixer1.Status.StandStill AND Mixer2.Status.StandStill THEN
			//
			// Calculate offset mixer 1 to mixer 2
			IF (f_ActPositionMixer1Calc + f_OffsetMixer1Mixer2) > 360 THEN
				fb_Mixer2.f_Position := f_ActPositionMixer1Calc + f_OffsetMixer1Mixer2 - 360;
			ELSE	
				fb_Mixer2.f_Position := f_ActPositionMixer1Calc + f_OffsetMixer1Mixer2;
			END_IF
			
			n_Step := 80;		
		END_IF
	
		//
		// Not Enable or Error	
		IF NOT b_Enable THEN
			n_Step := 10;
 		ELSIF b_ErrorInt THEN
			n_Step := 200;
		END_IF

	80:
		//
		//
		n_Step := 85;
		
		//
		// Not Enable or Error	
		IF NOT b_Enable THEN
			n_Step := 10;
 		ELSIF b_ErrorInt THEN
			n_Step := 200;
		END_IF
		
	85:
		//
		//
		IF fb_Mixer2.b_MoveAbsoluteDone THEN
			n_Step := 100;
		END_IF		
			
		//
		// Not Enable or Error	
		IF NOT b_Enable THEN
			n_Step := 10;
 		ELSIF b_ErrorInt THEN
			n_Step := 200;
		END_IF

	100:
		//
		// Couple
		IF fb_MC_GearIn.InGear THEN
			n_Step := 110;
		END_IF;
		
		//
		// Not Enable or Error
		IF NOT b_Enable THEN
			n_Step := 10;
 		ELSIF b_ErrorInt THEN
			n_Step := 200;
		END_IF	
	
	110:
		//
		//  Jog command possible (Coupled) via b_JogForward/b_JogBackwards
		
		
		//
		// Go to mode set position
		IF b_ModeSetPosition THEN
			n_Step := 20;	
		END_IF
		
		//
		// Not Enable or Error
		IF NOT b_Enable THEN
			n_Step := 10;
 		ELSIF b_ErrorInt THEN
			n_Step := 200;
		END_IF		
						
	200:
		// 	
		// GearOut
		IF fb_MC_GearOut.Done THEN
			n_Step := 210;
		END_IF
	
	210:
		//
		// No Error		
		IF NOT b_ErrorInt AND (b_Reset or not b_Enable) THEN
			n_Step := 10;
		END_IF
		
END_CASE


//
// Errors
b_ErrorInt:= fb_Mixer1.b_Error OR fb_Mixer2.b_Error OR fb_MC_GearIn.Error OR fb_MC_GearOut.Error;


//
// Outputs
b_PowerActiveMixer1			:= fb_Mixer1.b_PowerActive;
b_PowerActiveMixer2			:= fb_Mixer2.b_PowerActive;
b_ReadyToDrive				:= n_Step = 110;
b_ErrorGen					:= b_ErrorInt;
b_ErrorMixer1				:= fb_Mixer1.b_Error;
b_ErrorMixer2				:= fb_Mixer2.b_Error;
n_ErrorIDMixer1				:= fb_Mixer1.n_ErrorID;
n_ErrorIDMixer2				:= fb_Mixer2.n_ErrorID;
f_ActVelocityMixer1			:= fb_Mixer1.f_ActVelocity;
f_ActVelocityMixer2			:= fb_Mixer2.f_ActVelocity;
f_ActTorqueMixer1			:= fb_Mixer1.f_ActTorque;
f_ActTorqueMixer2			:= fb_Mixer2.f_ActTorque;
f_ActPositionMixer1			:= fb_Mixer1.f_ActPosition;
f_ActPositionMixer2			:= fb_Mixer2.f_ActPosition;
	
 
//
// Set position for mode SetPosition
IF n_Step = 30 THEN
	fb_Mixer1.f_Position := f_SetPositionMixer1;		
	fb_Mixer2.f_Position := f_SetPositionMixer2;
END_IF

//		
// Set velocity for Mixer 1/2		
IF n_Step = 110 THEN  
	fb_Mixer1.f_Velocity := f_Velocity;		   
	fb_Mixer2.f_Velocity := f_Velocity;	
ELSE
	fb_Mixer1.f_Velocity := 10;		   
	fb_Mixer2.f_Velocity := 10;
	f_Override:=100;
END_IF	   

//
// FB Mixer1
fb_Mixer1(
	Axis 					:= Mixer1,
	b_Enable 				:= b_Enable AND n_Step >= 35 AND n_Step <= 110,
	b_Reset					:= b_Reset AND NOT b_Enable,
	b_JogForward			:= (n_Step = 60 AND b_Mixer1InCollision) OR (n_Step = 110 AND b_JogForward),	  
	b_JogBackwards			:= (n_Step = 50 AND b_Mixer1InCollision) OR (n_Step = 110 AND b_JogBackwards),	
	b_MoveAbsolute			:= FALSE,
	n_MoveAbsoluteDirection := MC_Shortest_Way,
	b_Home					:= n_Step = 30 AND b_SetPositionMixer1,
	f_Acceleration			:= 0,
	f_Deceleration			:= 0,	
	f_Jerk					:= 0,
	f_Override 				:= f_Override);

	
//
// FB Mixer2
fb_Mixer2(
	Axis 					:= Mixer2,
	b_Enable 				:= b_Enable AND n_Step >= 35 AND n_Step <= 110,
	b_Reset					:= b_Reset AND NOT b_Enable,
	b_JogForward			:= (n_Step = 50 AND b_Mixer2InCollision),  
	b_JogBackwards			:= (n_Step = 60 AND b_Mixer2InCollision),	
	b_MoveAbsolute			:= n_Step = 80 OR n_Step = 85,
	n_MoveAbsoluteDirection := MC_Shortest_Way,
	b_Home					:= n_Step = 30 AND b_SetPositionMixer2,
	f_Acceleration			:= 0,
	f_Deceleration			:= 0,	
	f_Jerk					:= 0,
	f_Override 				:= f_Override);

//
// FB GearIn	
fb_MC_GearIn(
	Master 					:= Mixer1,
	Slave					:= Mixer2,
	Execute					:= b_Enable AND (n_Step = 100),
	RatioNumerator 			:= 1,
	RatioDenominator 		:= 1);
	                    	
//                      	
// FB GearOut           	
fb_MC_GearOut(          	
	Slave 					:= Mixer2,
	Execute					:= n_Step = 20 OR n_Step = 200);

END_FUNCTION_BLOCK

// ---- POUs/P_ModeSelector.TcPOU
PROGRAM P_ModeSelector
VAR
	
END_VAR

//***********************************************************************************
//
// ETH Zürich / Robotic Fabrication Lab
// HIB C 13 / Stefano-Franscini-Platz 1
// CH-8093 Zürich
// 
// ***********************************************************************************
// 
// PROJECT     :  A061 Digital Casting System
// 
// FUNCTION    :  selector for mode control
// 
// AUTHOR      :  Weiting Chen
// 
// EMAIL       :  
// 
// Copyright   : 
//
// ***********************************************************************************


GVL_VAR.b_Mode_Manual := GVL_IO.ib_CC1_Button_Mode_Manual;
GVL_VAR.b_Mode_Laptop := GVL_IO.ib_CC1_Button_Mode_Laptop;

END_PROGRAM

// ---- POUs/P_Set_Research_Data.TcPOU
PROGRAM P_Set_Research_Data
VAR


END_VAR

//***********************************************************************************
//
// ETH Zürich / Robotic Fabrication Lab
// HIB C 13 / Stefano-Franscini-Platz 1
// CH-8093 Zürich
// 
// ***********************************************************************************
// 
// PROJECT     :  A061 Inline Mixer
// 
// FUNCTION    :  Set all research data for the process
// 
// AUTHOR      :  Seyma Gürel / Philippe Fleischmann / Weiting Chen
// 
// EMAIL       :  scotto@arch.ethz.ch / fleischmann@arch.ehtz.ch
// 
// Copyright   :  ETH Zürich (CH) 2021
//
// ***********************************************************************************


//
// Updating Mixer 1 max speed [°/s]
GVL_ResearchData.f_RED_Control_Speed:=720;
GVL_VAR.f_MI1_MaxSpeed:=GVL_ResearchData.f_RED_Control_Speed;


//
// Updating Superplasticizer Pump checking values (WT 220916
GVL_ResearchData.n_RED_Superplasticizer_Pump_Check_Flowrate:=9;           // [ml/min]
GVL_ResearchData.n_RED_Superplasticizer_Pump_Check_Duration:=T#60000MS;   // [ms]
//GVL_ResearchData.f_RED_Superplasticizer_Pump_Density:=342.0;                    // [g/min]
GVL_ResearchData.f_RED_Superplasticizer_Pump_Density:=1.06;               // [g/cm^3]
GVL_ResearchData.n_RED_Superplasticizer_Pump_Flush_Speed:=GVL_ResearchData.f_RED_Status_Superplasticizer_Pump_Max_Flowrate_ml_per_min;		  // [ml/min]
//[32767 is equal 10v output and it means maximum setup speed from ViscoTech 654 rpm]


//
// Updating Acceleration Pump checking values (WT 220928
GVL_ResearchData.n_RED_Acceleration_Pump_Check_Flowrate:=90;     		// [ml/min]
GVL_ResearchData.n_RED_Acceleration_Pump_Check_Duration:=T#60000MS;   	// [ms]
//GVL_ResearchData.f_RED_Acceleration_Pump_Mass:=342.0;                    // [g/min]
GVL_ResearchData.f_RED_Acceleration_Pump_Density:=2.047;               // [g/cm^3]
GVL_ResearchData.n_RED_Acceleration_Pump_Flush_Speed:=GVL_ResearchData.f_RED_Status_Acceleration_Pump_Max_Flowrate_ml_per_min;

END_PROGRAM

// ---- POUs/P_SP1_Check.TcPOU
PROGRAM P_SP1_Check
VAR_INPUT
	//
	//INT
	n_Step: INT:=0;
END_VAR
VAR
	//
	// BOOL 
	b_Condition: BOOL;
	b_No_Emergency_Stop: BOOL:=TRUE;

	//
	// Timer
	t_SP1_Calibration_Time: TON; 
END_VAR

//***********************************************************************************
//
// ETH Zürich / Robotic Fabrication Lab
// HIB C 13 / Stefano-Franscini-Platz 1
// CH-8093 Zürich
// 
// ***********************************************************************************
// 
// PROJECT     :  A061 
// 
// FUNCTION    :  Step chain for Superplasticizer pump system check
// 
// AUTHOR      :  Weiting Chen / Philippe Fleischmann
// 
// EMAIL       :  
// 
// Copyright   :  
//
// ***********************************************************************************

//
// Ignore emergency stop
b_No_Emergency_Stop:=TRUE;

//
// Initalization
IF n_Step=0 THEN
	//
	// Check condition 
	b_Condition:=TRUE;
	//
	// Do 
	IF b_Condition THEN
		b_Condition:=FALSE;
		n_Step:=10;
	END_IF
END_IF

//
// Wait for activating calibration
IF n_Step=10 THEN
	//
	// Check condition 
	b_Condition:= GVL_ResearchData.b_RED_Superplasticizer_Pump_Check_On;
	//
	// Do
	IF b_Condition THEN
		b_Condition:=FALSE;
		n_Step:=20;
	END_IF
END_IF

//
// Wait for start 
IF n_Step=20 THEN
	//
	// Check condition 
	b_Condition:= GVL_IO.ib_SP1_Ready AND GVL_IO.ib_SP1_Button_On;
	//
	// Do 
	IF b_Condition THEN
		b_Condition:=FALSE;
		n_Step:=30;
	END_IF
END_IF

//
// Run calibration until time is over 
IF n_Step=30 THEN
	//
	// Check condition 
	b_Condition:=t_SP1_Calibration_Time.Q; 
	//
	// Do step
	IF b_Condition THEN
		b_Condition:=FALSE;
		n_Step:=40;
	END_IF
END_IF

//
// Reserve
IF n_Step=40 THEN
	//
	// Check condition 
	b_Condition:=TRUE;
	//
	// Do step
	IF b_Condition AND b_No_Emergency_Stop THEN
		b_Condition:=FALSE;
		n_Step:=50;
	END_IF
END_IF

//
// Return to step 10 
IF n_Step=50 THEN
	//
	// Check condition 
	b_Condition:=TRUE;
	//
	// Do step
	IF b_Condition THEN
		b_Condition:=FALSE;
		//
		// Reset calibrarion on
		GVL_ResearchData.b_RED_Superplasticizer_Pump_Check_On:=FALSE;
		n_Step:=10;
	END_IF
END_IF

// ****************************************
// Timer
// ****************************************
t_SP1_Calibration_Time(
	IN:=n_Step=30,
	PT:=GVL_ResearchData.n_RED_Superplasticizer_Pump_Check_Duration);

// ****************************************
// Reset
// ****************************************
IF NOT GVL_ResearchData.b_RED_Superplasticizer_Pump_Check_On THEN
  //
  // Rest step chain
  n_Step:=0;
END_IF

END_PROGRAM

// ---- POUs/P_SP1_OnOff.TcPOU
PROGRAM P_SP1_OnOff
VAR_INPUT
	//
	// INT
	n_step: INT := 0;
END_VAR
VAR	
	//
	// BOOL
	b_Condition: BOOL;
	b_No_Emergency_Stop:BOOL :=TRUE;
	
END_VAR

//***********************************************************************************
//
// ETH Zürich / Robotic Fabrication Lab
// HIB C 13 / Stefano-Franscini-Platz 1
// CH-8093 Zürich
// 
// ***********************************************************************************
// 
// PROJECT     :  A061 
// 
// FUNCTION    :  Step chain for Superplasticizer pump on or off 
// 
// AUTHOR      :  Weiting Chen / Philippe Fleischmann
// 
// EMAIL       :  
// 
// Copyright   :  
//
// ***********************************************************************************

//
// Ignore the emergency stop
b_No_Emergency_Stop:= TRUE;

//
// Initalization
IF n_Step=0 THEN
	//
	// Check condition 
	b_Condition:=TRUE;
	//
	// Do 
	IF b_Condition THEN
		b_Condition:=FALSE;
		n_Step:=10;
	END_IF
END_IF

//
// Wait for start mixer
IF n_Step=10 THEN
	//
	// Check condition 
	b_Condition:=GVL_IO.ib_SP1_Ready AND GVL_IO.ib_SP1_Button_On;
	//
	// Do 
	IF b_Condition AND b_No_Emergency_Stop THEN
		b_Condition:=FALSE;
		n_Step:=20;
	END_IF
END_IF

//
// Reserve
IF n_Step=20 THEN
	//
	// Check condition 
	b_Condition:=TRUE;
	//
	// Do 
	IF b_Condition AND b_No_Emergency_Stop THEN
		b_Condition:=FALSE;
		n_Step:=30;
	END_IF
END_IF

//
// Run for mixer 
IF n_Step=30 THEN
	//
	// Check condition 
	b_Condition:= NOT GVL_IO.ib_SP1_Button_Not_Off OR NOT GVL_IO.ib_SP1_No_Error;
	//
	// Do
	IF b_Condition THEN
		b_Condition:=FALSE;
		n_Step:=40;
	END_IF
END_IF

//
// Reserve
IF n_Step=40 THEN
	//
	// Check condition 
	b_Condition:=TRUE;
	//
	// Do 
	IF b_Condition AND b_No_Emergency_Stop THEN
		b_Condition:=FALSE;
		n_Step:=50;
	END_IF
END_IF

//
// Return to step 10 
IF n_Step=50 THEN
	//
	// Check condition 
	b_Condition:=TRUE;
	//
	// Do 
	IF b_Condition THEN
		b_Condition:=FALSE;
		n_Step:=10;
	END_IF
END_IF


//
// Write global variables
//

//
// Mixer run
GVL_VAR.b_SP1_Run:=n_step=30;

END_PROGRAM

// ---- POUs/P_AP1_Check.TcPOU
PROGRAM P_AP1_Check
VAR_INPUT
	//
	// INT 
	n_Step: INT := 0;	
END_VAR
VAR
	//
	// BOOL 
	b_Condition: BOOL;

	//
	// Timer
	t_AP1_Calibration_Time: TON; 
	
END_VAR

//***********************************************************************************
//
// ETH Zürich / Robotic Fabrication Lab
// HIB C 13 / Stefano-Franscini-Platz 1
// CH-8093 Zürich
// 
// ***********************************************************************************
// 
// PROJECT     :  A061 Inline Mixer
// 
// FUNCTION    :  Step chain for accelerator pump calibration
// 
// AUTHOR      :  Seyma Gürel / Philippe Fleischmann / Weiting Chen
// 
// EMAIL       :  sguerel@ethz.ch / fleischmann@arch.ehtz.ch
// 
// Copyright   :  ETH Zürich (CH) 2021
//
// ***********************************************************************************

//
// Initalization
IF n_Step=0 THEN
	//
	// Check condition 
	b_Condition:=TRUE;
	//
	// Do step
	IF b_Condition THEN
		b_Condition:=FALSE;
		n_Step:=10;
	END_IF
END_IF

//
// Wait for activating calibration
IF n_Step=10 THEN
	//
	// Check condition 
	b_Condition:= GVL_ResearchData.b_RED_Acceleration_Pump_Check_On;
	//
	// Do step
	IF b_Condition THEN
		b_Condition:=FALSE;
		n_Step:=20;
	END_IF
END_IF

//
// Wait for start 
IF n_Step=20 THEN
	//
	// Check condition 
	b_Condition:=GVL_IO.ib_AP1_Ready AND GVL_IO.ib_AP1_Button_On;
	//
	// Do step
	IF b_Condition THEN
		b_Condition:=FALSE;
		n_Step:=30;
	END_IF
END_IF

//
// Run calibration until time is over 
IF n_Step=30 THEN
	//
	// Check condition 
	b_Condition:=t_AP1_Calibration_Time.Q; 
	//
	// Do step
	IF b_Condition THEN
		b_Condition:=FALSE;
		n_Step:=40;
	END_IF
END_IF

//
// Return to step 10 
IF n_Step=40 THEN
	//
	// Check condition 
	b_Condition:=TRUE;
	//
	// Do step
	IF b_Condition THEN
		b_Condition:=FALSE;
		//
		// Reset calibrarion on
		GVL_ResearchData.b_RED_Acceleration_Pump_Check_On:=FALSE;
		n_Step:=10;
	END_IF
END_IF

// ****************************************
// Timer
// ****************************************
t_AP1_Calibration_Time(
	IN:=n_Step=30,
	PT:=GVL_ResearchData.n_RED_Acceleration_Pump_Check_Duration);

// ****************************************
// Reset
// ****************************************

IF NOT GVL_ResearchData.b_RED_Acceleration_Pump_Check_On THEN
  //
  // Rest step chain
  n_Step:=0;
END_IF

END_PROGRAM

// ---- POUs/P_Outputs_Manual.TcPOU
PROGRAM P_Outputs_Manual
VAR
	//
	//
	n_temp_speed_SP1: REAL;
	n_temp_speed_AP1: REAL;
	
END_VAR

//***********************************************************************************
//
// ETH Zürich / Robotic Fabrication Lab
// HIB C 13 / Stefano-Franscini-Platz 1
// CH-8093 Zürich
// 
// ***********************************************************************************
// 
// PROJECT     :  A061 Inline Mixer
// 
// FUNCTION    :  Outputs Manual Mode
// 
// AUTHOR      :  Fabio Scotto / Philippe Fleischmann / Weiting Chen
// 
// EMAIL       :  scotto@arch.ethz.ch / fleischmann@arch.ehtz.ch
// 
// Copyright   :  ETH Zürich (CH) 2020
//
// ***********************************************************************************


//***********************************************************************************
// Superplasticizer pump 1
//***********************************************************************************
//
// WT (220916)


//
// Power on
GVL_IO.ob_SP1_Power_On:=GVL_IO.ib_CC1_Button_Mode_Manual;
//
// Pressure is Okay, always set it to True
GVL_IO.ob_SP1_Pressure_Ok:=TRUE;
//
// Bucket is not empty, always set it to true
GVL_IO.ob_SP1_Not_Empty:=TRUE;
//
// Pulse mode is a preset amount,  not in use
GVL_IO.ob_SP1_Pulse:=FALSE;


//
// Start pump
IF		P_SP1_OnOff.n_step= 30 
	OR 	P_SP1_Check.n_Step= 30 
THEN
	//
	// Pump On
	GVL_IO.ob_SP1_Start:=TRUE;
ELSE
	//
	// Pump On
	GVL_IO.ob_SP1_Start:=FALSE;
END_IF

//
// Speeds for Superplastizier pump
IF GVL_ResearchData.b_RED_Superplasticizer_Pump_Flush_On AND P_SP1_OnOff.n_step= 30 THEN
	//
	// Process speed for flushing or filling the pipe
	n_temp_speed_SP1:=GVL_ResearchData.n_RED_Superplasticizer_Pump_Flush_Speed;

ELSIF P_SP1_Check.n_Step=20 OR P_SP1_Check.n_Step=30 THEN 	
	//	
	// Check Flowrate for pump
	n_temp_speed_SP1:=GVL_ResearchData.n_RED_Superplasticizer_Pump_Check_Flowrate;
	
ELSE
	//
	// Process speed for pump
	n_temp_speed_SP1:=GVL_ResearchData.n_RED_Superplasticizer_Pump_Flowrate;

END_IF

GVL_IO.on_SP1_Speed:=F_ScalAnalogOut(
	n_Input:= REAL_TO_INT(n_temp_speed_SP1),
	n_InMin:= 0, 
	n_InMax:= REAL_TO_INT(GVL_ResearchData.f_RED_Status_Superplasticizer_Pump_Max_Flowrate_ml_per_min), 
	n_OutMin:= 0, 
	n_OutMax:= 32767);


//***********************************************************************************
// Accelerator pump 1
//***********************************************************************************

//
// Power on
GVL_IO.ob_AP1_Power_On:=GVL_IO.ib_CC1_Button_Mode_Manual;
//
// Pressure okey always set to true
GVL_IO.ob_AP1_Pressure_Ok:=TRUE;
//
// Bucket not empty always set to true
GVL_IO.ob_AP1_Not_Empty:=TRUE;
//
// Pulse a preset amount not in use
GVL_IO.ob_AP1_Pulse:=FALSE;

//
// Start pump
IF 	   P_AP1_OnOff.n_Step=30 
	OR P_AP1_Check.n_Step=30
THEN
	//
	// Pump on
	GVL_IO.ob_AP1_Start:=TRUE;
ELSE
	//
	// Pump off
	GVL_IO.ob_AP1_Start:=FALSE;
END_IF

//
// Speed for accelerator pump
IF GVL_ResearchData.b_RED_Acceleration_Pump_Flush_On AND P_AP1_OnOff.n_Step=30 THEN
	//
	// Process speed for flushing or filling the pipe
	n_temp_speed_AP1:=GVL_ResearchData.n_RED_Acceleration_Pump_Flush_Speed;
ELSIF P_AP1_Check.n_Step=20 OR P_AP1_Check.n_Step=30 THEN
	//	
	// Check Flowrate for pump
	n_temp_speed_AP1:=GVL_ResearchData.n_RED_Acceleration_Pump_Check_Flowrate;
ELSE
	//
	// Process speed for pump
	n_temp_speed_AP1:=GVL_ResearchData.n_RED_Acceleration_Pump_Flowrate;
END_IF

GVL_IO.on_AP1_Speed:=F_ScalAnalogOut(
	n_Input:= REAL_TO_INT(n_temp_speed_AP1),
	n_InMin:= 0, 
	n_InMax:= REAL_TO_INT(GVL_ResearchData.f_RED_Status_Acceleration_Pump_Max_Flowrate_ml_per_min), 
	n_OutMin:= 0, 
	n_OutMax:= 32767);


// ***********************************************************************************
// Concrete Pump 1 
// ***********************************************************************************

//
// Start
IF  P_CP1_Enable.n_Step=20 THEN
	GVL_IO.ob_CP1_Start:=TRUE;
ELSE
	GVL_IO.ob_CP1_Start:=FALSE;
END_IF

//
// Stop
IF  P_CP1_Enable.n_Step=40 THEN
	GVL_IO.ob_CP1_Stop:=TRUE;
ELSE
	GVL_IO.ob_CP1_Stop:=FALSE;
END_IF

//
// Forward
GVL_IO.ob_CP1_Forward:=GVL_ResearchData.b_RED_Concrete_Pump_Forward_On;

//
// Backward
GVL_IO.ob_CP1_Backward:=GVL_ResearchData.b_RED_Concrete_Pump_Backward_On;

//
// Concrete pump speed  0 (0V) to 75 rpm (10V)
GVL_IO.on_CP1_Speed:=F_ScalAnalogOut(
	n_Input:=GVL_ResearchData.n_RED_Concrete_Pump_Speed, 
	n_InMin:=0, 
	n_InMax:=75, 
	n_OutMin:=0, 
	n_OutMax:=32767);

END_PROGRAM

// ---- POUs/P_Read_Research_Data.TcPOU
PROGRAM P_Read_Research_Data
VAR


END_VAR

//***********************************************************************************
//
// ETH Zürich / Robotic Fabrication Lab
// HIB C 13 / Stefano-Franscini-Platz 1
// CH-8093 Zürich
// 
// ***********************************************************************************
// 
// PROJECT     :  A061 Inline Mixer
// 
// FUNCTION    :  Read all research data for the process
// 
// AUTHOR      :  Seyma Gürel / Philippe Fleischmann
// 
// EMAIL       :  scotto@arch.ethz.ch / fleischmann@arch.ehtz.ch
// 
// Copyright   :  ETH Zürich (CH) 2021
//
// ***********************************************************************************

// 
// Mode [] (0916 WT)
GVL_ResearchData.b_RED_Mode_Manual:= GVL_VAR.b_Mode_Manual;
GVL_ResearchData.b_RED_Mode_Laptop:= GVL_VAR.b_Mode_Laptop;

//
// Mixer run []
GVL_ResearchData.b_RED_Status_On:=GVL_VAR.b_MI1_Run;

//
// Mixer 1 speed override [%]
GVL_ResearchData.f_RED_Status_Speed_Overide:=GVL_VAR.f_MI1_Override;

//
// Mixer 1 current speed []
GVL_ResearchData.f_RED_Status_Speed_Motor_1:=GVL.Axis_Mixer1.NcToPlc.ActVelo;

//
// Mixer 1 current torque []
GVL_ResearchData.f_RED_Status_Torque_Motor_1:=GVL.f_MID1_ActTorque;

//
// Mixer 1 current motor temperature []
GVL_ResearchData.f_RED_Status_Temperature_Motor_1:=GVL.in_MID1_ActMotorTemperature *0.1; // weiting added 220817

//
// Mixer 2 current speed []
GVL_ResearchData.f_RED_Status_Speed_Motor_2:=GVL.Axis_Mixer1.NcToPlc.ActVelo;

//
// Mixer 2 current torque []
GVL_ResearchData.f_RED_Status_Torque_Motor_2:=GVL.f_MID2_ActTorque;

//
// Mixer 1 current motor temperature []
GVL_ResearchData.f_RED_Status_Temperature_Motor_2:=GVL.in_MID2_ActMotorTemperature *0.1; // weiting added 220817


// Superplasticizer maximum pump flowrate [ml/min]
GVL_ResearchData.f_RED_Status_Superplasticizer_Pump_Max_Flowrate_ml_per_min:=18.0;

//
// Accelration pump flowrate [ml/min]
GVL_ResearchData.f_RED_Status_Acceleration_Pump_Max_Flowrate_ml_per_min:=180.0;

END_PROGRAM

// ---- POUs/P_CP1_Calibration.TcPOU
PROGRAM P_CP1_Calibration
VAR
END_VAR

//***********************************************************************************
//
// ETH Zürich / Robotic Fabrication Lab
// HIB C 13 / Stefano-Franscini-Platz 1
// CH-8093 Zürich
// 
// ***********************************************************************************
// 
// PROJECT     :  A061 
// 
// FUNCTION    :  Step chain for Concrete pump calibration
// 
// AUTHOR      :  Weiting Chen / Philippe Fleischmann
// 
// EMAIL       :  
// 
// Copyright   :  
//
// ***********************************************************************************
//
// placeholder for concrete pump calibration

END_PROGRAM
